// TwinCAT 3 PLC project GetDeviceData
// Title: GetDeviceData
// Company: Zeugwerk GmbH
// Author: Matthias Seehauser
// ProjectVersion: 1.0.0.0
// ProgramVersion: 3.1.4024.0
// libraries:
//   Tc2_IoFunctions, 3.4.4.0 (Beckhoff Automation GmbH)
//   Tc2_Standard, * (Beckhoff Automation GmbH)
//   Tc2_System, * (Beckhoff Automation GmbH)
//   Tc2_Utilities, * (Beckhoff Automation GmbH)
//   Tc3_Module, * (Beckhoff Automation GmbH)
//   ZCore, 1.6.0.3 (Zeugwerk GmbH)
// project tree:
//   / GetDeviceData.TcPOU, GetDeviceDataSteps.TcDUT, Parameter.TcGVL

// ---- GetDeviceDataSteps.TcDUT
{attribute 'qualified_only'}
TYPE GetDeviceDataSteps :
(
	Begin,
  FetchDeviceTypes,
  ResetId1,
  GetDeviceNames,
  ResetId2,
  GetDeviceNetIds,
  End
);
END_TYPE

// ---- Parameter.TcGVL
{attribute 'qualified_only'}
VAR_GLOBAL CONSTANT
  MaxDevicesSearchCount : UINT := 200;
  MaxDeviceToBeFound : UINT := 10;
END_VAR

// ---- GetDeviceData.TcPOU
{attribute 'no_explicit_call'}
{attribute 'conditionalshow_all_locals'}
FUNCTION_BLOCK GetDeviceData EXTENDS ZCore.Object IMPLEMENTS ZCore.IUnmanagedObject
VAR_OUTPUT
  NameArray : ARRAY[0..Parameter.MaxDeviceToBeFound] OF ZCore.ZString;
  NetIdArray : ARRAY[0..Parameter.MaxDeviceToBeFound] OF Tc2_System.T_AmsNetID;
END_VAR
VAR
  _amsNetId : Tc2_System.T_AmsNetID;
  _ethercatMasterCount : UINT;
  _step : ZCore.Step(GetDeviceDataSteps.Begin, GetDeviceDataSteps.End);
END_VAR

/// The cyclic method should be run in any PLC-cycle. If the object has no work to do, we will simply
/// RETURN here. If an action has been started, this cyclic method takes care of all the work to do.
METHOD Cyclic
VAR_INST
  itIndex : UINT;
  ethercatMasters : UINT;
  indexArray : ARRAY[0..Parameter.MaxDeviceToBeFound] OF UINT;

  getDeviceType : Tc2_IoFunctions.IOF_GetDeviceType;
  getDeviceName : Tc2_IoFunctions.IOF_GetDeviceName;
  getDeviceNetIds : Tc2_IoFunctions.IOF_GetDeviceNetId;
END_VAR
CASE _step.Index OF
  GetDeviceDataSteps.Begin:
    IF Busy
    THEN
      _ethercatMasterCount := 0;
      _step.SetNext(GetDeviceDataSteps.FetchDeviceTypes);
    END_IF
  
  GetDeviceDataSteps.FetchDeviceTypes:
    IF _step.OnEntry()
    THEN
      getDeviceType(START:=FALSE);
      getDeviceType(START:=TRUE, NETID:=_amsNetId, DEVICEID:=ItIndex, TMOUT:=T#2S);
    END_IF
    
    getDeviceType(START:=FALSE);
    IF getDeviceType.ERR // no valid device found
    THEN
      IF ItIndex > Parameter.MaxDevicesSearchCount 
      THEN
        _step.SetNext(GetDeviceDataSteps.ResetId1);
      ELSE
        _step.SetNext(GetDeviceDataSteps.FetchDeviceTypes);
      END_IF
      
      itIndex := itIndex + 1;
    ELSIF NOT getDeviceType.BUSY
    THEN
      IF getDeviceType.IODeviceType = Tc2_IoFunctions.IODEVICETYPE_ETHERCAT
      THEN
        IndexArray[_ethercatMasterCount] := itIndex;
        _ethercatMasterCount := _ethercatMasterCount + 1;
        itIndex := itIndex + 1;
        _step.SetNext(GetDeviceDataSteps.ResetId1);
      END_IF
    END_IF

  GetDeviceDataSteps.ResetId1:
    itIndex := 0;
    _step.SetNext(GetDeviceDataSteps.GetDeviceNames);  
    
  GetDeviceDataSteps.GetDeviceNames:
    IF _step.OnEntry()
    THEN
      getDeviceName(START:=FALSE);
      getDeviceName(START:=TRUE, NETID:=_amsNetId, DEVICEID:=IndexArray[ItIndex], TMOUT:=T#2S);
    END_IF  
    
    getDeviceName();
    IF getDeviceName.ERR
    THEN
      Abort('Name could not be fetched!');
    ELSIF NOT getDeviceName.BUSY
    THEN
      NameArray[itIndex] := getDeviceName.DEVICENAME;
      itIndex := itIndex + 1;
      IF IndexArray[itIndex] <> 0
      THEN
        _step.SetNext(GetDeviceDataSteps.GetDeviceNames);
      ELSE
        _step.SetNext(GetDeviceDataSteps.ResetId2);
      END_IF
    END_IF
    
  GetDeviceDataSteps.ResetId2:
    itIndex := 0;
    _step.SetNext(GetDeviceDataSteps.GetDeviceNetIds);  
    
  GetDeviceDataSteps.GetDeviceNetIds:
    IF _step.OnEntry()
    THEN
      getDeviceNetIds(START:=FALSE);
      getDeviceNetIds(START:=TRUE, NETID:=_amsNetId, DEVICEID:=IndexArray[itIndex], TMOUT:=T#2S);
    END_IF  
    
    getDeviceNetIds();
    IF getDeviceNetIds.ERR
    THEN
      Abort('Name could not be fetched!');
    ELSIF NOT getDeviceNetIds.BUSY
    THEN
      NetIdArray[itIndex] := getDeviceNetIds.DeviceNetId;
      itIndex := itIndex + 1;
      IF IndexArray[itIndex] = 0
      THEN
        SetBusy(FALSE);
        _step.SetNext(GetDeviceDataSteps.End);
      END_IF
    END_IF      
  
  GetDeviceDataSteps.End:
    RETURN;
    
END_CASE
END_METHOD

/// Starts reading of all available Ethercat-Master Device names
/// Just wait until Busy property of this object returns FALSE -> then fetch all Ethercat Master names from
/// the Array in VAR_INPUT of this object
METHOD DeviceNamesAsync
VAR_INPUT
  amsNetId : Tc2_System.T_AmsNetID; //< AMS-Netid of the IPC on which the device names should be fetched
END_VAR
SetBusy(TRUE);
_amsNetId := amsNetId;
_step.SetNext(GetDeviceDataSteps.Begin);
END_METHOD

/// Returns the actual found Ethercat Master count -> Needed to iterate through the VAR_INPUT Arrays of AMSNet-IDs and
/// Ethercat Master Device names.
PROPERTY EthercatMasterCount : UINT
GET
EthercatMasterCount := _ethercatMasterCount;
END_GET
END_PROPERTY

/// Sets the object to Idle-State becuse no booting phase is needed here!
METHOD FB_init : BOOL
VAR_INPUT
	bInitRetains : BOOL; // if TRUE, the retain variables are initialized (warm start / cold start)
	bInCopyCode : BOOL;  // if TRUE, the instance afterwards gets moved into the copy code (online change)
END_VAR
SetIdle();
END_METHOD

END_FUNCTION_BLOCK
